Staubli VAL3: language.pgx

public program language()
  local num l_nWhich
begin
  //-----------------------------------------------------------------------
  //Header begin
  //Description of program
  //  This program lets you choose the language : English or Deutsch
  //
  //Traceability
  //  Creation : 07-04-08 - f.Rob
  //Header end
  //-----------------------------------------------------------------------
  userPage()
  cls()
  gotoxy(5,5)
  putln(sUsrMess[101])
  gotoxy(7,10)
  put(sUsrMess[0])
  //Functions to display navigation keys (F1 through F8)
  //(here F3 and F6 with messages "Germ" or "Engl")
  call usrButtonTxt(3,"Germ")
  call usrButtonTxt(6,"Engl")
  //Waiting user choice 3 (F3) or 6 (F6)
  do
    l_nWhich=(get()-270)
  until ((l_nWhich==3) or (l_nWhich==6))
  //User choice : 3 (F3)=> Deutsch, 6 (F6)=> English
  switch l_nWhich
    case 3
      nLangSet=0
    break
    case 6
      nLangSet=100
    break
  endSwitch
  cls()
  userPage()
  gotoxy(0,13)
  put("                                       ")
end
